// TIA Portal project "TicTacToe" (V17)

(* hardware
DEVICE "S7-1500/ET200MP station_1"  S7-1500 station
   slot 0: "Rail_0"  Rack  6ES7 590-1***0-0AA0
   slot 1: "PLC_1"  CPU 1515-2 PN  6ES7 515-2AM02-0AB0  V2.9
      slot 3: "CPU display_1"  6ES7591-1BA00-0AA0
      slot 32768: "PROFINET interface_1"  X1
         slot 32769: "Port_1"  X1 P1
         slot 32770: "Port_2"  X1 P2
      slot 33024: "PROFINET interface_2"  X2
         slot 33025: "Port_1"  X2 P1
      slot 34817: "Virtual CP interface port_1"  Virtual CP interface port  Virtual CP interface port
DEVICE "HMI_1"  TP1500 Comfort
   slot 0: "HMI_1"  TP1500 Comfort  6AV2 124-0QC02-0AX0  17.0.0.0
   slot 1: "HMI_RT_1"  TP1500 Comfort  6AV2 124-0QC02-0AX0  17.0.0.0
   slot 5: "HMI_1.IE_CP_1"  PROFINET Interface  17.0.0.0
      slot 1: "PROFINET Interface_1"  PROFINET Interface
         slot 1: "Port_1"  Port
         slot 2: "Port_2"  Port
   slot 6: "HMI_1.IE_CP_2"  PROFINET Interface  17.0.0.0
      slot 1: "PROFINET Interface_GBit"  PROFINET Interface
         slot 1: "Port_1"  Port
   slot 7: "HMI_1.MPI/DP_CP_1"  MPI/DP Interface  17.0.0.0
*)

// ===== PLC "PLC_1"  CPU 1515-2 PN =====

TYPE "GameField_PLCD"
   STRUCT
      state : Int;
      xFree : Bool := true;
      xPressed : Bool;
   END_STRUCT;
END_TYPE

TYPE "LeaderBoardEntry_PLCD"
   STRUCT
      "Name" : WString;
      TurnsToWin : Int;
      "Date" : LDT;
   END_STRUCT;
END_TYPE

TYPE "AIScore"
   STRUCT
      score : Int;
      row : Int;
      col : Int;
   END_STRUCT;
END_TYPE

DATA_BLOCK "MainDB"   // DB1
{ S7_Optimized_Access := 'TRUE' }
VERSION : 0.1
   VAR
      xResetGame : Bool;   // Resets the Game Board
      GameState : Struct
         xGameOver : Bool;
         xGameHasWinner : Bool;
         xGameIsDraw : Bool;
         iGameWinner : Int;
         iTurns : Int;
      END_STRUCT;
      PlayerMode : Int := 1;
      Player : Struct
         Names : Struct
            Player_1 : WString := WSTRING#'X';
            Player_2 : WString := WSTRING#'O';
         END_STRUCT;
         CurrentTurn : Int := 1;
         LastTurn : Int := 1;
      END_STRUCT;
      Difficulty : Int := 1;
   END_VAR
   VAR RETAIN
      GameBoard : Array[1..3, 1..3] of "GameField_PLCD";
      GameBoardAI : Array[1..3, 1..3] of "GameField_PLCD";
   END_VAR
   VAR
      GameBoardEmpty : "GameField_PLCD";
      xResetAIScore : Bool;
      AIScores : Array[0..50] of "AIScore";
      AIScoreEmpy : "AIScore";
      LeaderBoard : Array[0..10] of "LeaderBoardEntry_PLCD";
      LeaderBoardEmpty : "LeaderBoardEntry_PLCD";
      xResetLeaderBoard : Bool;
   END_VAR
BEGIN
   GameBoardEmpty.xFree := true;
   GameBoardEmpty.xPressed := false;
   GameBoardEmpty.state := 0;
END_DATA_BLOCK

DATA_BLOCK "FBMain_DB"   // DB2
{ S7_Optimized_Access := 'TRUE' }
VERSION : 0.1
// stored: InstanceOfName FBMain
"FBMain"
BEGIN
END_DATA_BLOCK

FUNCTION_BLOCK "FBMain"   // FB1, FBD
{ S7_Optimized_Access := 'TRUE' }
VERSION : 0.1
   VAR
      Edges : Array[0..10] of Bool;
      NextMove : Bool;
      MoveTo : Array[0..1] of Int;
      PEdge : R_TRIG;
   END_VAR
   VAR_TEMP
      ModePVP : Bool;
      ModeKI : Bool;
      DifficultyEasy : Bool;
      DifficultyHard : Bool;
      DifficultyInsane : Bool;
      i : Int;
      k : Int;
      player : Int;
      xDrawDetect : Bool;
      WinningPlayer : Int;
      BestScore : Int;
      Score : Int;
      RandomRow : UDInt;
      RandomCol : UDInt;
      RandomError : Bool;
      RandomStatus : Word;
      RandomSubStatus : Word;
      "Date" : LDT;
      RetVal : Int;
   END_VAR
   VAR CONSTANT
      X : Int := 1;
      O : Int := 2;
      PVP : Int := 1;
      AI : Int := 2;
      Human : Int := 1;
      Empty : Int;
      Player_1 : Int := 1;
      Player_2 : Int := 2;
      NegativeMax : Int := -32768;   // Highest possible Negative score Int16 :)
      PositiveMax : Int := 32767;   // Highest possible Positive Number in Int16 :)
      Easy : Int := 1;   // Game Difficulty
      Hard : Int := 2;   // Game Difficulty
      Insane : Int := 3;   // Game Difficulty
   END_VAR
   // MoveTo[0] := 1;
   // MoveTo[1] := 1;
   // // Edges[0] : Edge GameField any Pressed
BEGIN

REGION Network 1
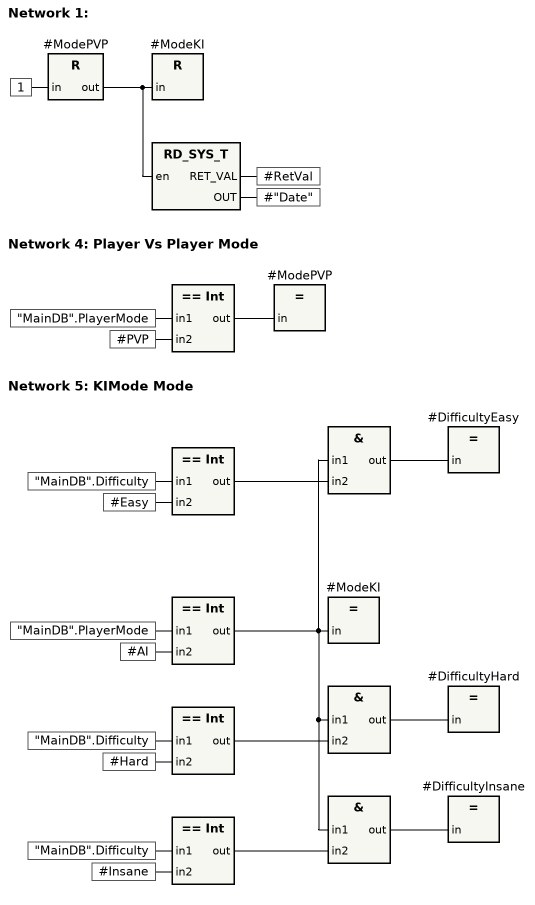
   IF 1 THEN
       #ModePVP := FALSE;
       #ModeKI := FALSE;
       #RetVal := RD_SYS_T(OUT => #"Date");
   END_IF;
END_REGION

REGION Network 2 (SCL): Reset GameBoard
   IF "MainDB".xResetGame THEN
       // Reset GameField
       FOR #k := 1 TO 3 DO
           FOR #i := 1 TO 3 DO
               "MainDB".GameBoard[#k, #i] := "MainDB".GameBoardEmpty;
           END_FOR;
       END_FOR;

       FOR #i := 0 TO 50 DO
           "MainDB".AIScores[#i] := "MainDB".AIScoreEmpy;
       END_FOR;
       //Reset Current Player to 1 
       "MainDB".Player.CurrentTurn := 1;
       "MainDB".GameState.xGameOver := false;
       "MainDB".GameState.xGameHasWinner := false;
       "MainDB".GameState.xGameIsDraw := false;
       "MainDB".GameState.iGameWinner := 0;
       "MainDB".xResetGame := 0;
       "MainDB".GameState.iTurns := 0;
   END_IF;
END_REGION

REGION Network 3 (SCL): Reset AI Score For Debugging
   IF "MainDB".xResetAIScore THEN
       // Remove all AI Debugging Scores
       FOR #i := 0 TO 50 DO
           "MainDB".AIScores[#i] := "MainDB".AIScoreEmpy;
       END_FOR;
       "MainDB".xResetAIScore := 0;
   END_IF;
END_REGION

REGION Network 4: Player Vs Player Mode
   #ModePVP := "MainDB".PlayerMode = #PVP;
END_REGION

REGION Network 5: KIMode Mode
   #ModeKI := "MainDB".PlayerMode = #AI;
   #DifficultyEasy := #ModeKI AND ("MainDB".Difficulty = #Easy);
   #DifficultyHard := #ModeKI AND ("MainDB".Difficulty = #Hard);
   #DifficultyInsane := #ModeKI AND ("MainDB".Difficulty = #Insane);
END_REGION

REGION Network 6 (SCL): PVPMode = GameBoardLogic
   IF #ModePVP THEN
       FOR #k := 1 TO 3 DO
           FOR #i := 1 TO 3 DO
               IF "MainDB".GameBoard[#k,#i].xPressed = 1 AND "MainDB".GameBoard[#k,#i].xFree = 1 THEN

                   // Update LastPlayer with Current Player
                   "MainDB".Player.LastTurn := "MainDB".Player.CurrentTurn;
                   "MainDB".GameBoard[#k, #i].state := "MainDB".Player.CurrentTurn;

                   // Update The CurrentPlayer
                   CASE "MainDB".Player.CurrentTurn OF
                       1:"MainDB".Player.CurrentTurn := 2; // Player 1 -> Player 2
                       3:"MainDB".Player.CurrentTurn := 1; // Player 2 -> Player 1
                       ELSE  // Statement section ELSE
                           "MainDB".Player.CurrentTurn := 1; // Player 0 -> Player 1
                   END_CASE;

                   "MainDB".GameBoard[#k, #i].xFree := 0;
                   "MainDB".GameBoard[#k, #i].xPressed := 0;


               END_IF;
           END_FOR;
       END_FOR;
   END_IF;
END_REGION

REGION Network 7 (SCL): KIMode [Easy] = GameBoardLogic
   IF #ModeKI AND #DifficultyEasy THEN
       CASE "MainDB".Player.CurrentTurn OF
           #O:  // Human Will Play
               FOR #k := 1 TO 3 DO
                   FOR #i := 1 TO 3 DO
                       IF "MainDB".GameBoard[#k, #i].xPressed = 1 AND "MainDB".GameBoard[#k, #i].xFree = 1 THEN
                           "MainDB".Player.LastTurn := "MainDB".Player.CurrentTurn;
                           "MainDB".GameBoard[#k, #i].state := #O;
                           "MainDB".Player.CurrentTurn := #X; // Next Move is AI Turn
                           "MainDB".GameBoard[#k, #i].xFree := 0;
                           "MainDB".GameBoard[#k, #i].xPressed := 0;
                           "MainDB".GameState.iTurns := "MainDB".GameState.iTurns + 1;
                       END_IF;
                   END_FOR;
               END_FOR;
           #X:  // Dumb AI Will Play
               FOR #k := 1 TO 3 DO
                   FOR #i := 1 TO 3 DO
                       IF "MainDB".GameBoard[#k, #i].state = 0 AND "MainDB".GameBoard[#k, #i].xFree = 1 THEN
                           // Actual Make our Move
                           "MainDB".Player.LastTurn := "MainDB".Player.CurrentTurn;
                           "MainDB".GameBoard[#k, #i].state := #X;
                           "MainDB".GameBoard[#k, #i].xFree := 0;
                           "MainDB".Player.CurrentTurn := #O;
                           "MainDB".GameState.iTurns := "MainDB".GameState.iTurns + 1;
                           EXIT;
                       END_IF;
                   END_FOR;
                   IF "MainDB".Player.CurrentTurn = #O OR "MainDB".GameState.xGameOver THEN
                       EXIT;
                   END_IF;
               END_FOR;
       END_CASE;
   END_IF;
END_REGION

REGION Network 8 (SCL): KIMode [Hard] = GameBoardLogic
   IF #ModeKI AND #DifficultyHard THEN
       CASE "MainDB".Player.CurrentTurn OF
            #O:  // Human Will Play
               FOR #k := 1 TO 3 DO
                   FOR #i := 1 TO 3 DO
                       IF "MainDB".GameBoard[#k, #i].xPressed = 1 AND "MainDB".GameBoard[#k, #i].xFree = 1 THEN
                           "MainDB".Player.LastTurn := "MainDB".Player.CurrentTurn;
                           "MainDB".GameBoard[#k, #i].state :=#O;
                           "MainDB".Player.CurrentTurn := #X; // Next Move is AI Turn
                           "MainDB".GameBoard[#k, #i].xFree := 0;
                           "MainDB".GameBoard[#k, #i].xPressed := 0;
                           "MainDB".GameState.iTurns := "MainDB".GameState.iTurns + 1;
                       END_IF;
                   END_FOR;
               END_FOR;
           #X:  // Dumb AI Will Play
               REPEAT
                   #RandomRow := "LGF_RandomRange_UDInt"(minValue := 1, maxValue := 3, error=>#RandomError, status=>#RandomStatus, subfunctionStatus=>#RandomSubStatus);
                   #RandomCol :="LGF_RandomRange_UDInt"(minValue:=1, maxValue:=3, error=>#RandomError, status=>#RandomStatus, subfunctionStatus=>#RandomSubStatus);
                   #k := UDINT_TO_INT(#RandomRow);
                   #i := UDINT_TO_INT(#RandomCol);
                   IF "MainDB".GameBoard[#k, #i].state = 0 AND "MainDB".GameBoard[#k, #i].xFree = 1 THEN
                       "MainDB".Player.LastTurn := "MainDB".Player.CurrentTurn;
                       "MainDB".GameBoard[#k, #i].state := #X;
                       "MainDB".GameBoard[#k, #i].xFree := 0;
                       "MainDB".Player.CurrentTurn := #O;
                       "MainDB".GameState.iTurns := "MainDB".GameState.iTurns + 1;
                   END_IF;
               UNTIL "MainDB".Player.CurrentTurn = #O OR "MainDB".GameState.xGameOver END_REPEAT;

       END_CASE;
   END_IF;
END_REGION

REGION Network 9 (SCL): KIMode [Insane] = GameBoardLogic
   IF #ModeKI AND #DifficultyInsane THEN

       CASE "MainDB".Player.CurrentTurn OF
           1:  //Player 1 will be AI
               #BestScore := #NegativeMax;
               "MainDB".GameBoardAI := "MainDB".GameBoard;
               FOR #k := 1 TO 3 DO
                   FOR #i := 1 TO 3 DO
                       IF "MainDB".GameBoard[#k, #i].state = 0 THEN
                           "MainDB".GameBoard[#k, #i].state := #X;
                           #Score := "MiniMax"(BoardState := "MainDB".GameBoard, depth := 0, isMaximizing := FALSE);
                           "AiScoreManager"(Score := #Score,
                                            Row := #k,
                                            Col := #i);
                           "MainDB".GameBoard[#k, #i].state := #Empty;
                           IF #Score > #BestScore THEN
                               #BestScore := #Score;
                               #MoveTo[0] := #k;
                               #MoveTo[1] := #i;
                           END_IF;
                       END_IF;
                   END_FOR;
               END_FOR;
               // Actual Make our Move
               "MainDB".Player.LastTurn := "MainDB".Player.CurrentTurn;
               "MainDB".GameBoard[#MoveTo[0], #MoveTo[1]].state := #X;
               "MainDB".GameBoard[#MoveTo[0], #MoveTo[1]].xFree := 0;
               "MainDB".Player.CurrentTurn := #O;
               "MainDB".GameState.iTurns := "MainDB".GameState.iTurns + 1;
           2:  // Ai Will Play
               FOR #k := 1 TO 3 DO
                   FOR #i := 1 TO 3 DO
                       IF "MainDB".GameBoard[#k, #i].xPressed = 1 AND "MainDB".GameBoard[#k, #i].xFree = 1 THEN
                           "MainDB".Player.LastTurn := "MainDB".Player.CurrentTurn;
                           "MainDB".GameBoard[#k, #i].state := #O;
                           "MainDB".Player.CurrentTurn := #X; // Next Move is AI Turn
                           "MainDB".GameBoard[#k, #i].xFree := 0;
                           "MainDB".GameBoard[#k, #i].xPressed := 0;
                           "MainDB".GameBoardAI := "MainDB".GameBoard;
                           "MainDB".GameState.iTurns := "MainDB".GameState.iTurns + 1;
                       END_IF;
                   END_FOR;
               END_FOR;

       END_CASE;

   END_IF;
END_REGION

REGION Network 10 (SCL): Winner
   #WinningPlayer :="Winner"( "MainDB".GameBoard);
   CASE #WinningPlayer OF
       0:  // Game is still Ongoing
           ;
       1..2: // Player 1 or 2 Won
           "MainDB".GameState.xGameOver := true;
           "MainDB".GameState.xGameHasWinner := true;
           "MainDB".GameState.iGameWinner := #WinningPlayer;

       3: // Game has a Draw
           "MainDB".GameState.xGameOver := true;
           "MainDB".GameState.xGameIsDraw := true;
   END_CASE;
END_REGION

REGION Network 11 (SCL): LeaderBoard

   #PEdge(CLK:="MainDB".GameState.xGameOver AND "MainDB".GameState.xGameHasWinner,
          Q=>#Edges[1]);

   IF #Edges[1] THEN
       CASE #WinningPlayer OF
           1:  // Statement section case 1
               "LeaderBoard"(Name := "MainDB".Player.Names.Player_1,
                             TurnsToWin := "MainDB".GameState.iTurns,
                             "Date" := #Date);

           2:  // Statement section case 2 to 4
               "LeaderBoard"(Name := "MainDB".Player.Names.Player_2,
                             TurnsToWin := "MainDB".GameState.iTurns,
                             "Date" := #Date);
       END_CASE;
   END_IF;

   IF "MainDB".xResetLeaderBoard THEN
       FOR #i := 0 TO 10 DO
           "MainDB".LeaderBoard[#i] := "MainDB".LeaderBoardEmpty;
       END_FOR;
       "MainDB".xResetLeaderBoard := false;
   END_IF;
END_REGION

REGION Network 12 (SCL): Look Board if Game is Over
   IF "MainDB".GameState.xGameOver THEN
       FOR #i := 1 TO 3 DO
           FOR #k := 1 TO 3 DO
               "MainDB".GameBoard[#i, #k].xFree := false;
           END_FOR;
       END_FOR;


   END_IF;
END_REGION
END_FUNCTION_BLOCK

FUNCTION "MiniMax" : Int   // FC1, SCL
{ S7_Optimized_Access := 'TRUE' }
VERSION : 0.1
   VAR_INPUT
      depth : Int;   // The Depth of the Board we are Checking
      isMaximizing : Bool;   // False => Human Player | True => AI
   END_VAR
   VAR_IN_OUT
      BoardState : Array[1..3, 1..3] of "GameField_PLCD";
   END_VAR
   VAR_TEMP
      i : Int;   // Rows
      k : Int;   // Colums
      BestScore : Int;
      Score : Int;
      Winner : Int;   // 0=> Game Not Over. 1/2 => Won Player 1/2, 3=> Draw
   END_VAR
   // Ret_Val : Best Score
   VAR CONSTANT
      NegativeMax : Int := -32768;   // Highest possible Negative Number in Int16 :)
      PositiveMax : Int := 32767;   // Highest possible Positive Number in Int16 :)
      X : Int := 1;
      O : Int := 2;
      Score_X : Int := 10;
      Score_O : Int := -10;
      Score_Draw : Int;
   END_VAR
BEGIN
   REGION Winner
       #Winner := "Winner"(#BoardState);
       IF #Winner <> 0 THEN
           CASE #Winner OF
               1:#BestScore := #Score_X;
               2:#BestScore := #Score_O;
               3:#BestScore := #Score_Draw;
               ELSE
                   #BestScore := #Score_Draw;
           END_CASE;
           #MiniMax := #BestScore;
           RETURN;
       END_IF;
   END_REGION


   REGION MaxiMizing
       //Maximizing Value
       IF #isMaximizing = TRUE THEN
           #BestScore := #NegativeMax;
           FOR #i := 1 TO 3 DO
               FOR #k := 1 TO 3 DO
                   IF #BoardState[#i, #k].state = 0 THEN
                       #BoardState[#i, #k].state := #X;
                       #Score := "MiniMax"(BoardState := #BoardState, depth := #depth + 1, isMaximizing := FALSE);
                       #BoardState[#i, #k].state := 0;
                       #BestScore := MAX(IN1 := #Score, IN2 := #BestScore);
                   END_IF;
               END_FOR;
           END_FOR;
           #MiniMax := #BestScore;
           RETURN;
       END_IF;
   END_REGION

   REGION MiniMizing
       IF #isMaximizing = FALSE THEN
           #BestScore := #PositiveMax;
           FOR #i := 1 TO 3 DO
               FOR #k := 1 TO 3 DO
                   IF #BoardState[#i, #k].state = 0 THEN
                       #BoardState[#i, #k].state := #O;
                       #Score := "MiniMax"(BoardState := #BoardState, depth := #depth + 1, isMaximizing := TRUE);
                       #BoardState[#i, #k].state := 0;
                       #BestScore := MIN(IN1 := #Score, IN2 := #BestScore);
                   END_IF;
               END_FOR;
           END_FOR;
           #MiniMax := #BestScore;
           RETURN;
       END_IF;
   END_REGION

   //Just Here since the retarded Compiler cannot figure out the above Logic
   #MiniMax := 0;
END_FUNCTION

FUNCTION "Winner" : Int   // FC2, SCL
{ S7_Optimized_Access := 'TRUE' }
VERSION : 0.1
   VAR_IN_OUT
      BoardState : Array[1..3, 1..3] of "GameField_PLCD";   // State of our current Board
   END_VAR
   VAR_TEMP
      i : Int;   // Loop Counter
      k : Int;   // Loop Counter
      xHasFreeSpots : Bool;
   END_VAR
   // Ret_Val : 0=> Game Not Over. 1/2 => Won Player 1/2, 3=> Draw
   VAR CONSTANT
      Draw : Int := 3;
   END_VAR
BEGIN
   REGION Initialize
       // Statement section REGION
       #Winner := 0;
   END_REGION


   REGION Horizontal Condition
       FOR #i := 1 TO 3 DO
           // Check for 0 States we don't want to evaluate them
           IF     "MainDB".GameBoard[#i, 1].state = 0
               OR "MainDB".GameBoard[#i, 1].state = 0
               OR "MainDB".GameBoard[#i, 1].state = 0 THEN
               CONTINUE; // next Loop
           END_IF;

            //Evaluate Winning Condition Horizontal
           (*
           ---------------|
             X  |  X | X  |
           ---------------|
                |    |    |
           ---------------|
                |    |    |
           ---------------|
           *)
           IF      "MainDB".GameBoard[#i, 1].state = "MainDB".GameBoard[#i, 2].state
               AND "MainDB".GameBoard[#i, 2].state = "MainDB".GameBoard[#i, 3].state
               AND "MainDB".GameBoard[#i, 1].state = "MainDB".GameBoard[#i, 3].state THEN
               #Winner := "MainDB".GameBoard[#i, 1].state;
               RETURN; // Leave Block No Farther Evaluation needed
           END_IF;
       END_FOR;
   END_REGION


   REGION Vertical Condition
       FOR #i := 1 TO 3 DO
           // Check for 0 States we don't want to evaluate them
           IF "MainDB".GameBoard[1,#i].state = 0
               OR "MainDB".GameBoard[1,#i].state = 0
               OR "MainDB".GameBoard[1,#i].state = 0 THEN
               CONTINUE; // next Loop
           END_IF;

           //Evaluate Winning Condition Vertical
           (*
           ---------------|
             X  |    |    |
           ---------------|
             X  |    |    |
           ---------------|
             X  |    |    |
           ---------------|
           *)
           IF "MainDB".GameBoard[1,#i].state = "MainDB".GameBoard[2,#i].state
               AND "MainDB".GameBoard[2,#i].state = "MainDB".GameBoard[3,#i].state
               AND "MainDB".GameBoard[1,#i].state = "MainDB".GameBoard[3,#i].state THEN
               #Winner := "MainDB".GameBoard[1,#i].state;
               RETURN; // Leave Block No Farther Evaluation needed
           END_IF;
       END_FOR;
   END_REGION


   REGION Diagonal
       // Check for 0 States we don't want to evaluate them
       IF "MainDB".GameBoard[1, 1].state <> 0
           OR "MainDB".GameBoard[2,2].state <> 0
           OR "MainDB".GameBoard[3, 3].state <> 0 THEN

           // Diagonal Win Check
           (*
           ---------------|
            X   |    |    |
           ---------------|
                | X  |    |
           ---------------|
               |    |  X  |
           ---------------|
           *)
           IF "MainDB".GameBoard[1, 1].state = "MainDB".GameBoard[2, 2].state
               AND "MainDB".GameBoard[2, 2].state = "MainDB".GameBoard[3, 3].state
               AND "MainDB".GameBoard[1, 1].state = "MainDB".GameBoard[3, 3].state THEN
               #Winner := "MainDB".GameBoard[1, 1].state;
               RETURN; // Leave Block No Farther Evaluation needed
           END_IF;
       END_IF;
   END_REGION

   REGION Diagonal Oposed
       // Check for 0 States we don't want to evaluate them
       IF "MainDB".GameBoard[1, 3].state <> 0
           OR "MainDB".GameBoard[2, 2].state <> 0
           OR "MainDB".GameBoard[3, 1].state <> 0 THEN

           //  Oposite Across Win Check
           (*
           ---------------|
                |    | X  |
           ---------------|
                | X  |    |
           ---------------|
            X   |    |    |
           ---------------|
           *)
           IF "MainDB".GameBoard[1, 3].state = "MainDB".GameBoard[2, 2].state
               AND "MainDB".GameBoard[2, 2].state = "MainDB".GameBoard[3, 1].state
               AND "MainDB".GameBoard[1, 3].state = "MainDB".GameBoard[3, 1].state THEN
               #Winner := "MainDB".GameBoard[1, 3].state;
               RETURN; // Leave Block No Farther Evaluation needed
           END_IF;
       END_IF;
   END_REGION

   REGION Detect a Draw
       //Detect Draw (Simple Way)
       #xHasFreeSpots := FALSE;
       FOR #i := 1 TO 3 DO
           FOR #k := 1 TO 3 DO // Statement section FOR
               IF "MainDB".GameBoard[#i, #k].state = 0 THEN
                   #xHasFreeSpots := TRUE;
               END_IF;
           END_FOR;
       END_FOR;

       IF #xHasFreeSpots = FALSE THEN
           #Winner := #Draw;
           RETURN;
       END_IF;
   END_REGION
END_FUNCTION

FUNCTION "AiScoreManager" : Void   // FC3, SCL
{ S7_Optimized_Access := 'TRUE' }
VERSION : 0.1
   VAR_INPUT
      Score : Int;
      Row : Int;
      Col : Int;
   END_VAR
   VAR_TEMP
      i : Int;   // Loop Counter
   END_VAR
BEGIN
   REGION SaveAndRotate
       FOR #i := 50 TO 1 BY -1 DO
           "MainDB".AIScores[#i] := "MainDB".AIScores[#i - 1];
       END_FOR;
       "MainDB".AIScores[0].score := #Score;
       "MainDB".AIScores[0].row := #Row;
       "MainDB".AIScores[0].col := #Col;
   END_REGION
END_FUNCTION

FUNCTION "LeaderBoard" : Void   // FC7, SCL
{ S7_Optimized_Access := 'TRUE' }
VERSION : 0.1
   VAR_INPUT
      "Name" : WString;
      TurnsToWin : Int;
      "Date" : LDT;
   END_VAR
   VAR_TEMP
      i : Int;   // Loop
   END_VAR
BEGIN
   REGION SaveAndRotate
       FOR #i := 10 TO 1 BY -1 DO
           "MainDB".LeaderBoard[#i] := "MainDB".LeaderBoard[#i - 1];
       END_FOR;
       "MainDB".LeaderBoard[0].Name := #Name;
       "MainDB".LeaderBoard[0].TurnsToWin := #TurnsToWin;
       "MainDB".LeaderBoard[0]."Date" := #Date;
   END_REGION
END_FUNCTION

ORGANIZATION_BLOCK "Main"   // OB1, LAD, ProgramCycle
TITLE = "Main Program Sweep (Cycle)"
{ S7_Optimized_Access := 'TRUE' }
VERSION : 0.1
   VAR_INPUT
      Initial_Call : Bool;   // Initial call of this OB
      Remanence : Bool;   // =True, if remanent data are available
   END_VAR
   VAR_TEMP
      Result : Int;
   END_VAR
BEGIN

REGION Network 1: GameLogic
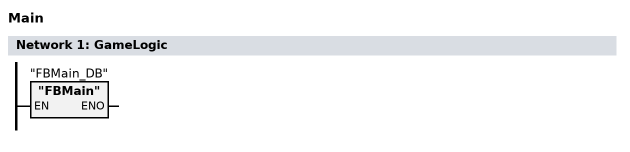
   RUNG wire#powerrail
      "FBMain_DB"()
   END_RUNG
   // the same network as SCL:
   "FBMain_DB"();   // "FBMain"
END_REGION
END_ORGANIZATION_BLOCK

// folder: FC_TEST

FUNCTION "FC1" : Void   // FC4, FBD
{ S7_Optimized_Access := 'TRUE' }
VERSION : 0.1
   VAR_TEMP
      Temp : Int;
   END_VAR
BEGIN

REGION Network 1
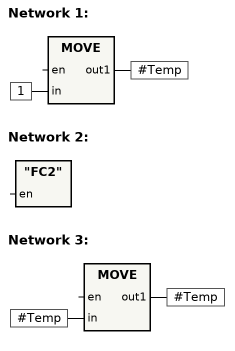
   #Temp := 1;
END_REGION

REGION Network 2
   "FC2"();
END_REGION

REGION Network 3
   #Temp := #Temp;
END_REGION
END_FUNCTION

FUNCTION "FC2" : Void   // FC5, FBD
{ S7_Optimized_Access := 'TRUE' }
VERSION : 0.1
   VAR_TEMP
      Temp : Int;
   END_VAR
BEGIN

REGION Network 1
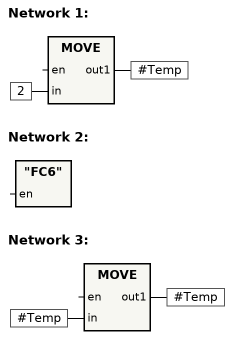
   #Temp := 2;
END_REGION

REGION Network 2
   "FC6"();
END_REGION

REGION Network 3
   #Temp := #Temp;
END_REGION
END_FUNCTION

FUNCTION "FC6" : Void   // FC6, FBD
{ S7_Optimized_Access := 'TRUE' }
VERSION : 0.1
   VAR_TEMP
      Temp : Int;
   END_VAR
BEGIN

REGION Network 1
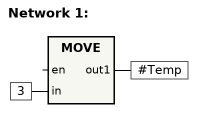
   #Temp := 3;
END_REGION
END_FUNCTION

// folder: LGF

FUNCTION "LGF_RandomRange_UDInt" : UDInt   // FC10079, SCL
TITLE = LGF_RandomRange_UDInt
{ S7_Optimized_Access := 'TRUE' }
AUTHOR : Siemens_Digital_Industries
FAMILY : LGF
NAME : LGF_RandomRange_UDInt
// This function generates random numbers in defined limits (Datatype UDInt)
   VAR_INPUT
      minValue : UDInt;   // minimal Value random can reach / Minimum value of the range of the random number
      maxValue : UDInt;   // maximal Value random can reach / Maximum value of the range of the random number
   END_VAR
   VAR_OUTPUT
      error : Bool;   // Error if true
      status : Word;   // Status of the function
      subfunctionStatus : Word;   // Status or return value of called FB's, FCs and system blocks
   END_VAR
   VAR_TEMP
      tempTime : DTL;   // System time
      tempNanoSecondInDWord : DWord;   // UDINT converted to DWORD for access to individual bytes
      tempTimeStatus : Word;   // Status of the instruction RD_SYS_T
      tempRandomValue : DWord;   // Random-start-value
      tempNormReal : Real;   // Normalized value
   END_VAR
   // Ret_Val : Returns random UDInt number in a predefined range
   VAR CONSTANT
      ZERO : UDInt := 0;   // Zero value in case of error
      MAX_UDINT : UDInt := 4294967295 ;   // Maximum UDINT value
      SUB_STATUS_NO_ERROR : Word := 16#0000;   // Status: sub function call ends without error
      STATUS_FINISHED_NO_ERROR : Word := 16#0000;   // Status: Execution finished without errors
      ERR_MAX_LESS_MIN : Word := 16#8200;   // Error: The maximum limit number is smaller than the minimum limit number
      ERR_RD_SYS_T : Word := 16#8600;   // Error: System function Read system time returned an error
   END_VAR
BEGIN
   REGION Block info header
     //=============================================================================
     // SIEMENS AG / (c)Copyright 2019
     //-----------------------------------------------------------------------------
     // Title:            LGF_RandomRange_UDInt
     // Comment/Function: This function generates random numbers in defined limits (Datatype UDInt)
     // Library/Family:   LGF(Library General Functions)
     // Author:           Siemens Digital Industry Support
     // Tested with:      S7-PLCSIM Advanced V2.0 SP1
     // Engineering:      TIA Portal V15 Update 2
     // Restrictions:     ENO disabled - error handling done by error and status
     // Requirements:     PLC (S7-1200 / S7-1500)
     //-------------------------------------------------------------------------------
     // Change log table:
     // Version  | Date       | Expert in charge       | Changes applied
     //----------|------------|------------------------|------------------------------
     // 01.00.00 11.12.2019  Siemens Industry Online Support
     //                      First released version
     //                      copied from "LGF_RandomRange_DInt"
     // 03.00.00 23.04.2020  Siemens Industry Support
     //                      Set version to V3.0.0, harmonize the version of the whole library
     //=============================================================================
   END_REGION

   REGION Validation
     // Check if the maximal Value is less than the minimal value
     IF (#minValue > #maxValue) THEN
       #error := true;
       #status := #ERR_MAX_LESS_MIN;
       #subfunctionStatus := #SUB_STATUS_NO_ERROR;
       #LGF_RandomRange_UDInt := #ZERO;
       RETURN;
     END_IF;

     // Read system time
     #tempTimeStatus := INT_TO_WORD(RD_SYS_T(#tempTime));

     // Check return variable for error
     IF (#tempTimeStatus <> #SUB_STATUS_NO_ERROR) THEN
       #error := true;
       #status := #ERR_RD_SYS_T;
       #subfunctionStatus := #tempTimeStatus;
       #LGF_RandomRange_UDInt := #ZERO;
       RETURN;
     END_IF;
   END_REGION

   REGION Calculating random number
     // Converting to double word so individual bytes can be addressed
     #tempNanoSecondInDWord := UDINT_TO_DWORD(#tempTime.NANOSECOND);

     // Calculate a random-start-value depending on the time
     #tempRandomValue.%B3 := #tempNanoSecondInDWord.%B0;
     #tempRandomValue.%B2 := #tempNanoSecondInDWord.%B1;
     #tempRandomValue.%B1 := #tempNanoSecondInDWord.%B2;
     #tempRandomValue.%B0 := #tempNanoSecondInDWord.%B3;

     // Norm the calculated random number: 0.0 <= #tempNormReal <= 1.0
     #tempNormReal := UDINT_TO_REAL(DWORD_TO_UDINT(#tempRandomValue)) / UDINT_TO_REAL(#MAX_UDINT);

     // Scale the tempNormReal to be in the range of maxValue and minValue
     #LGF_RandomRange_UDInt := REAL_TO_UDINT((#tempNormReal * UDINT_TO_REAL(#maxValue - #minValue) + UDINT_TO_REAL(#minValue)));

     #error := false;
     #status := #STATUS_FINISHED_NO_ERROR;
     #subfunctionStatus := #SUB_STATUS_NO_ERROR;
     // ENO mechanism is not used
     ENO := TRUE;
   END_REGION
END_FUNCTION

(* ===== HMI "HMI_RT_1" =====
system functions are stored by id; their names below are inferred from use
connection "HMI_Connection_1": ETHERNET, S7_1500_OMS

HMI tags "Default tag table"
   "MainDB_PlayerMode" : Int = PLC MainDB.PlayerMode, 100 ms
   "MainDB_Difficulty" : Int = PLC MainDB.Difficulty, 100 ms
   "MainDB_CurrentTurn" : Int = PLC MainDB.Player.CurrentTurn, 100 ms
   "MainDB_Player_Names_Player_1" : WString[254] = PLC MainDB.Player.Names.Player_1, 100 ms
   "MainDB_Player_Names_Player_2" : WString[254] = PLC MainDB.Player.Names.Player_2, 100 ms
   "MainDB_xResetGame" : Bool = PLC MainDB.xResetGame, 100 ms
   "MainDB_Player_CurrentTurn" : Int = PLC MainDB.Player.CurrentTurn, 100 ms
   "MainDB_GameState_iGameWinner" : Int = PLC MainDB.GameState.iGameWinner, 100 ms
   "MainDB_GameState_xGameHasWinner" : Bool = PLC MainDB.GameState.xGameHasWinner, 100 ms
   "MainDB_GameState_xGameIsDraw" : Bool = PLC MainDB.GameState.xGameIsDraw, 1 s
   "MainDB_xResetAIScore" : Bool = PLC MainDB.xResetAIScore, 1 s
   "MainDB_LeaderBoard{0}" : LeaderBoardEntry_PLCD = PLC MainDB.LeaderBoard[0], 1 s
   "MainDB_LeaderBoard{1}" : LeaderBoardEntry_PLCD = PLC MainDB.LeaderBoard[1], 1 s
   "MainDB_LeaderBoard{2}" : LeaderBoardEntry_PLCD = PLC MainDB.LeaderBoard[2], 1 s
   "MainDB_LeaderBoard{3}" : LeaderBoardEntry_PLCD = PLC MainDB.LeaderBoard[3], 1 s
   "MainDB_LeaderBoard{4}" : LeaderBoardEntry_PLCD = PLC MainDB.LeaderBoard[4], 1 s
   "MainDB_LeaderBoard{5}" : LeaderBoardEntry_PLCD = PLC MainDB.LeaderBoard[5], 1 s
   "MainDB_LeaderBoard{6}" : LeaderBoardEntry_PLCD = PLC MainDB.LeaderBoard[6], 1 s
   "MainDB_LeaderBoard{7}" : LeaderBoardEntry_PLCD = PLC MainDB.LeaderBoard[7], 1 s
   "MainDB_LeaderBoard{8}" : LeaderBoardEntry_PLCD = PLC MainDB.LeaderBoard[8], 1 s
   "MainDB_LeaderBoard{9}" : LeaderBoardEntry_PLCD = PLC MainDB.LeaderBoard[9], 1 s
   "MainDB_LeaderBoard{10}" : LeaderBoardEntry_PLCD = PLC MainDB.LeaderBoard[10], 1 s
   "MainDB_xResetLeaderBoard" : Bool = PLC MainDB.xResetLeaderBoard, 1 s

HMI tags "GameBoard"
   "MainDB_GameBoard{1,1}" : GameField_PLCD = PLC MainDB.GameBoard[1,1], 100 ms
   "MainDB_GameBoard{1,2}" : GameField_PLCD = PLC MainDB.GameBoard[1,2], 100 ms
   "MainDB_GameBoard{1,3}" : GameField_PLCD = PLC MainDB.GameBoard[1,3], 100 ms
   "MainDB_GameBoard{2,1}" : GameField_PLCD = PLC MainDB.GameBoard[2,1], 100 ms
   "MainDB_GameBoard{2,2}" : GameField_PLCD = PLC MainDB.GameBoard[2,2], 100 ms
   "MainDB_GameBoard{2,3}" : GameField_PLCD = PLC MainDB.GameBoard[2,3], 100 ms
   "MainDB_GameBoard{3,1}" : GameField_PLCD = PLC MainDB.GameBoard[3,1], 100 ms
   "MainDB_GameBoard{3,2}" : GameField_PLCD = PLC MainDB.GameBoard[3,2], 100 ms
   "MainDB_GameBoard{3,3}" : GameField_PLCD = PLC MainDB.GameBoard[3,3], 100 ms

text list "PlayerType": 1 'PlayerVSPlayer'; 2 'PlayerVSKI'

text list "Diffculty": 1 'Easy'; 2 'Hard'; 3 'Insane'

text list "Turn": 1 'Player 1'; 2 'Player 2'; 3 'KI'

Template "Template_1" 1280x800
   Button "Exit" at 1200,739 size 78x59; TextOff 'Exit'; PictureOff "ExitRuntime_TP1500_Comfort_TR"; PictureOn "ExitRuntime_TP1500_Comfort_TR"
      on Release: StopRuntime(0)
   Button "Template_Button" at 1120,739 size 78x59; TextOff 'Text'
   Button "Template_Button_1" at 1040,739 size 78x59; TextOff 'Text'
   Button "Template_Button_2" at 960,739 size 78x59; TextOff 'Text'
   Button "Template_Button_3" at 880,739 size 78x59; TextOff 'Text'
   Button "Template_Button_4" at 800,739 size 78x59; TextOff 'Text'
   Button "Template_Button_5" at 720,739 size 78x59; TextOff 'Text'
   Button "Template_Button_6" at 640,739 size 78x59; TextOff 'Text'
   Button "Template_Button_7" at 561,739 size 78x59; TextOff 'Text'
   Button "Template_Button_8" at 481,739 size 78x59; TextOff 'Text'
   Button "Template_Button_9" at 401,739 size 78x59; TextOff 'Text'
   Button "Template_Button_10" at 321,739 size 78x59; TextOff 'Text'
   Button "Template_Button_11" at 241,739 size 78x59; TextOff 'Text'
   Button "Template_Button_12" at 161,739 size 78x59; TextOff 'Text'
   Button "Template_Button_13" at 81,739 size 78x59; TextOff 'Text'
   Button "Start screen" at 1,739 size 78x59; TextOff 'Start screen'; PictureOff "NavigateHome_TP1500_Comfort_TR"; PictureOn "NavigateHome_TP1500_Comfort_TR"
      on Release: ActivateScreen("Root screen", 0)

screen "Root screen" 1280x800, template "Template_1"
   SymbolicIOField "PlayerVsPlayer" at 126,77 size 197x32; TextOff '0'; TextOn '1'; TextList "PlayerType"
      ProcessValue <- "MainDB_PlayerMode"
      on Change: SetBit("MainDB_xResetGame")
   SymbolicIOField "Difficulty" at 126,114 size 197x32; TextOn '1'; TextOff '0'; TextList "Diffculty"
      ProcessValue <- "MainDB_Difficulty"
      Visibility <- "MainDB_PlayerMode"
      on Change: SetBit("MainDB_xResetGame")
   ScreenModuleView "GameField_1_1" at 392,216 size 150x150; ScreenModuleType ""
      Guid_{11997190-3471} <- "MainDB_GameBoard{1,1}"
   ScreenModuleView "GameField_1_2" at 554,216 size 150x150; ScreenModuleType ""
      Guid_{11997190-3471} <- "MainDB_GameBoard{1,2}"
   ScreenModuleView "GameField_1_3" at 716,216 size 150x150; ScreenModuleType ""
      Guid_{11997190-3471} <- "MainDB_GameBoard{1,3}"
   ScreenModuleView "GameField_2_1" at 391,380 size 150x150; ScreenModuleType ""
      Guid_{11997190-3471} <- "MainDB_GameBoard{2,1}"
   ScreenModuleView "GameField_2_2" at 554,380 size 150x150; ScreenModuleType ""
      Guid_{11997190-3471} <- "MainDB_GameBoard{2,2}"
   ScreenModuleView "GameField_2_3" at 716,380 size 150x150; ScreenModuleType ""
      Guid_{11997190-3471} <- "MainDB_GameBoard{2,3}"
   ScreenModuleView "GameField_3_1" at 392,544 size 150x150; ScreenModuleType ""
      Guid_{11997190-3471} <- "MainDB_GameBoard{3,1}"
   ScreenModuleView "GameField_3_2" at 554,544 size 150x150; ScreenModuleType ""
      Guid_{11997190-3471} <- "MainDB_GameBoard{3,2}"
   ScreenModuleView "GameField_3_3" at 716,544 size 150x150; ScreenModuleType ""
      Guid_{11997190-3471} <- "MainDB_GameBoard{3,3}"
   IOField "IO_Player1_Name" at 24,182 size 300x32; FormatPattern ??????????????????????????
      ProcessValue <- "MainDB_Player_Names_Player_1"
      Visibility <- "MainDB_PlayerMode"
   IOField "IO_Player2_Name" at 24,257 size 301x32; FormatPattern ??????????????????????
      ProcessValue <- "MainDB_Player_Names_Player_2"
   TextField "Label_Player1_Name" at 24,153 size 300x33; Text 'Player 1 Name:'
      Visibility <- "MainDB_PlayerMode"
   TextField "Label_Player2_Name" at 24,228 size 301x33; Text 'Player 2 Name:'
   Button "Button_1" at 41,306 size 268x32; TextOff 'Reset Game'
      on Release: SetBit("MainDB_xResetGame")
   TextField "Text field_1" at 513,57 size 250x47; Text 'Current Turn'
   SymbolicIOField "Symbolic I/O field_1" at 376,110 size 518x46; TextOff '0'; TextOn '1'; TextList "Turn"
      ProcessValue <- "MainDB_Player_CurrentTurn"
   ScreenModuleView "WinnerScreen_1" at 378,206 size 517x506; ScreenModuleType ""
      Guid_{11997190-5089} <- "MainDB_GameState_iGameWinner"
      Guid_{11997190-5245} <- "MainDB_Player_Names_Player_1"
      Guid_{11997190-5249} <- "MainDB_Player_Names_Player_2"
      Guid_{11997190-5098} <- "MainDB_GameState_xGameHasWinner"
      Guid_{11997190-6561} <- "MainDB_xResetGame"
   ScreenModuleView "DrawScreen_1" at 378,206 size 517x507; ScreenModuleType ""
      Guid_{11997190-6229} <- "MainDB_xResetGame"
      Guid_{11997190-5098} <- "MainDB_GameState_xGameIsDraw"
   Button "Button_2" at 41,489 size 268x32; TextOff 'Reset AI Score'
      on Release: SetBit("MainDB_xResetAIScore")
   TextField "Text field_2" at 22,22 size 319x37; Text 'TicTacToe GameMode'
   TextField "Text field_3" at 25,77 size 105x32; Text 'Mode'
   TextField "Text field_4" at 25,114 size 105x32; Text 'Difficulty'
   TextField "Text field_5" at 963,22 size 53x25; Text 'Info:'
   TextField "Text field_6" at 961,47 size 306x292; Text 'Player VS Player: In this Mode you Play against 2 Players and can Choice a Name PlayerVsAI: Easy = Linear Placement of X Hard = Random Placement on Board Insane = MiniMax Algo :) Good Luck Please let the AI Finish First Its not Locked yet. There are still some bugs feel free to fix them or let me know and i fix them s.Krumbach@hahnautomation.com'
   Button "Button_3" at 40,346 size 268x32; TextOff 'Leader Board'
      on Release: function_efd93a16("LeaderBoard", 378, 206, -1, -1, 1)

PopupScreen "LeaderBoard" 550x420
   ScreenModuleView "LeaderBoarrdEntry_1" at 9,22 size 512x32; ScreenModuleType ""
      Guid_{11997190-8529} <- "MainDB_LeaderBoard{0}"
   ScreenModuleView "LeaderBoarrdEntry_2" at 9,50 size 512x32; ScreenModuleType ""
      Guid_{11997190-8529} <- "MainDB_LeaderBoard{1}"
   ScreenModuleView "LeaderBoarrdEntry_3" at 9,78 size 512x32; ScreenModuleType ""
      Guid_{11997190-8529} <- "MainDB_LeaderBoard{2}"
   ScreenModuleView "LeaderBoarrdEntry_4" at 9,106 size 512x32; ScreenModuleType ""
      Guid_{11997190-8529} <- "MainDB_LeaderBoard{3}"
   ScreenModuleView "LeaderBoarrdEntry_5" at 9,134 size 512x32; ScreenModuleType ""
      Guid_{11997190-8529} <- "MainDB_LeaderBoard{4}"
   ScreenModuleView "LeaderBoarrdEntry_6" at 9,162 size 512x32; ScreenModuleType ""
      Guid_{11997190-8529} <- "MainDB_LeaderBoard{5}"
   ScreenModuleView "LeaderBoarrdEntry_7" at 9,190 size 512x32; ScreenModuleType ""
      Guid_{11997190-8529} <- "MainDB_LeaderBoard{6}"
   ScreenModuleView "LeaderBoarrdEntry_8" at 9,218 size 512x32; ScreenModuleType ""
      Guid_{11997190-8529} <- "MainDB_LeaderBoard{7}"
   ScreenModuleView "LeaderBoarrdEntry_9" at 9,246 size 512x32; ScreenModuleType ""
      Guid_{11997190-8529} <- "MainDB_LeaderBoard{8}"
   ScreenModuleView "LeaderBoarrdEntry_10" at 9,274 size 512x32; ScreenModuleType ""
      Guid_{11997190-8529} <- "MainDB_LeaderBoard{9}"
   ScreenModuleView "LeaderBoarrdEntry_11" at 9,302 size 512x32; ScreenModuleType ""
      Guid_{11997190-8529} <- "MainDB_LeaderBoard{10}"
   Button "Button_1" at 275,363 size 214x32; TextOff 'Close'
      on Activate: function_efd93a16("LeaderBoard", 0, 0, 0, -1, 1)
   Button "Button_2" at 47,363 size 189x32; TextOff 'Reset Leaderboard'
      on Activate: SetBit("MainDB_xResetLeaderBoard")
*)

(* ===== HMI "HMI_RT_1" =====
system functions are stored by id; their names below are inferred from use

HMI tags "Default tag table"
   "state" : Int, internal
   "xpressed" : Bool, internal

graphic list "State": 1 'circle'; 2 'cross'; 0 'none'

ScreenModuleEditorView "GameField" 640x480
   GraphicIOField "Graphic I/O field_1" at 10,10 size 100x100; PictureList "State"
      ProcessValue <- "PLCD_GameField.state"
   Button "Button_1" at 10,10 size 100x100; TextOff 'Text'
      on Activate: SetBit("PLCD_GameField.xPressed")
      ObjectEnable <- "PLCD_GameField.xFree"
*)

(* ===== HMI "HMI_RT_1" =====
system functions are stored by id; their names below are inferred from use

ScreenModuleEditorView "DrawScreen" 640x480
   Rectangle "Background" at 10,10 size 507x505
      Visibility <- "Visible"
   TextField "Headline" at 152,15 size 205x39; Text 'No Winner -.-'
      Visibility <- "Visible"
   Button "Button_1" at 90,165 size 332x148; TextOff 'I know i Can Win this... I Play again !!!'
      on Release: SetBit("PlayAgain")
      Visibility <- "Visible"
*)

(* ===== HMI "HMI_RT_1" =====
system functions are stored by id; their names below are inferred from use

text list "Turn": 1 'Player 1'; 2 'Player 2'; 3 'KI'

ScreenModuleEditorView "WinnerScreen" 640x480
   Rectangle "Background" at 10,10 size 507x505
      Visibility <- "Visible"
   TextField "Headline" at 184,20 size 154x39; Text 'Winner :)'
      Visibility <- "Visible"
   SymbolicIOField "WinnerName" at 99,62 size 324x41; TextOn '1'; TextOff '0'; TextList "Turn"
      ProcessValue <- "iWinner"
      Visibility <- "Visible"
   GraphicView "WinnerAnimation" at 32,112 size 463x387; Picture "Winner"
      Visibility <- "Visible"
   Button "Button_1" at 56,316 size 152x75; TextOff 'Play Again !!'
      Visibility <- "Visible"
      on Release: SetBit("btnPlayAgain")
*)

(* ===== HMI "HMI_RT_1" =====
system functions are stored by id; their names below are inferred from use

HMI tags "Default tag table"
   "state" : Int, internal
   "xpressed" : Bool, internal

graphic list "State": 2 'circle'; 1 'cross'; 0 'none'

ScreenModuleEditorView "GameField" 640x480
   GraphicIOField "Graphic I/O field_1" at 10,10 size 100x100; PictureList "State"
      ProcessValue <- "PLCD_GameField.state"
   Button "Button_1" at 10,10 size 100x100; TextOff 'Text'
      on Activate: SetBit("PLCD_GameField.xPressed")
      ObjectEnable <- "PLCD_GameField.xFree"
*)

(* ===== HMI "HMI_RT_1" =====

ScreenModuleEditorView "LeaderBoarrdEntry" 640x480
   IOField "I/O field_1" at 10,10 size 232x32; FormatPattern ????????????????????
   IOField "I/O field_2" at 238,10 size 39x32; FormatPattern 99
   IOField "I/O field_3" at 273,10 size 249x32; FormatPattern 9999999
*)

(* ===== HMI "HMI_RT_1" =====

ScreenModuleEditorView "LeaderBoarrdEntry" 640x480
   IOField "I/O field_1" at 10,10 size 232x32; FormatPattern ????????????????????
      ProcessValue <- "LeaderBoardEntry.Name"
   IOField "I/O field_2" at 238,10 size 39x32; FormatPattern 99
      ProcessValue <- "LeaderBoardEntry.TurnsToWin"
   IOField "I/O field_3" at 273,10 size 249x32; FormatPattern 9999999
      ProcessValue <- "LeaderBoardEntry.Date"
*)

(* ===== HMI "HMI_RT_1" =====
system functions are stored by id; their names below are inferred from use

HMI tags "Default tag table"
   "state" : Int, internal
   "xpressed" : Bool, internal

graphic list "State": 2 'circle'; 1 'cross'; 0 'none'

ScreenModuleEditorView "GameField" 640x480
   GraphicIOField "Graphic I/O field_1" at 10,10 size 100x100; PictureList "State"
      ProcessValue <- "PLCD_GameField.state"
   Button "Button_1" at 10,10 size 100x100; TextOff 'Text'
      ObjectEnable <- "PLCD_GameField.xFree"
      on Press: function_b14e0dd5("PLCD_GameField.xPressed", 0)
*)